FUNCTION_BLOCK DataTypesInteger (* Template for an empty basic function block *)
  (* Standard: 61499-2; Description: Normal just propagates the input to the output Max: sets to the highest possible value Min: sets to the lowest possible value Internal: sets the output from inside Copyright (c) 2019 Jan Holzweber This program and the accompanying materials are made available under the terms of the Eclipse Public License 2.0 which is available at https://www.eclipse.org/legal/epl-2.0/ SPDX-License-Identifier: EPL-2.0 *)
  (* Version 1.0, 2019-06-05, jholz *)
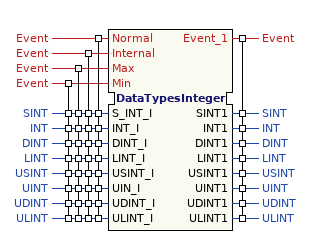
  EVENT_INPUT
    Normal WITH S_INT_I, INT_I, DINT_I, LINT_I, USINT_I, UIN_I, UDINT_I, ULINT_I;
    Internal WITH S_INT_I, INT_I, DINT_I, LINT_I, USINT_I, UIN_I, UDINT_I, ULINT_I;
    Max WITH S_INT_I, INT_I, DINT_I, LINT_I, USINT_I, UIN_I, UDINT_I, ULINT_I;
    Min WITH INT_I, S_INT_I, DINT_I, LINT_I, USINT_I, UIN_I, UDINT_I, ULINT_I;
  END_EVENT
  EVENT_OUTPUT
    Event_1 WITH SINT1, INT1, DINT1, LINT1, USINT1, UINT1, UDINT1, ULINT1;
  END_EVENT
  VAR_INPUT
    S_INT_I : SINT;
    INT_I : INT;
    DINT_I : DINT;
    LINT_I : LINT;
    USINT_I : USINT;
    UIN_I : UINT;
    UDINT_I : UDINT;
    ULINT_I : ULINT;
  END_VAR
  VAR_OUTPUT
    SINT1 : SINT;
    INT1 : INT;
    DINT1 : DINT;
    LINT1 : LINT;
    USINT1 : USINT;
    UINT1 : UINT;
    UDINT1 : UDINT;
    ULINT1 : ULINT;
  END_VAR
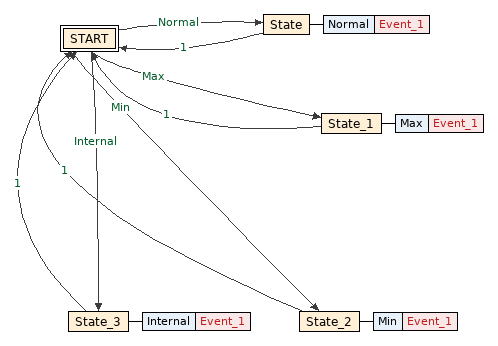
  EC_STATES
    START; (* Initial State *)
    State : Normal -> Event_1;
    State_1 : Max -> Event_1;
    State_2 : Min -> Event_1;
    State_3 : Internal -> Event_1;
  END_STATES
  EC_TRANSITIONS
    START TO State := Normal;
    State TO START := 1;
    START TO State_1 := Max;
    State_1 TO START := 1;
    START TO State_2 := Min;
    State_2 TO START := 1;
    START TO State_3 := Internal;
    State_3 TO START := 1;
  END_TRANSITIONS
  ALGORITHM Normal IN ST: (* new algorithm *)
SINT1 :=S_INT_I;
INT1:=INT_I;
DINT1:=DINT_I;
LINT1:=LINT_I;
USINT1:=USINT_I;
UINT1:=UIN_I;
UDINT1:=UDINT_I;
ULINT1:=ULINT_I;
  END_ALGORITHM
  ALGORITHM Max IN ST: (* new algorithm *)
SINT1 :=127;
INT1:=32767;
DINT1:=2147483647;
LINT1:=9223372036854775807;
USINT1:=255;
UINT1:=65535;
UDINT1:=4294967295;
ULINT1:=1;
  END_ALGORITHM
  ALGORITHM Min IN ST: (* new algorithm *)
SINT1 :=-128;
INT1:=-32768;
DINT1:=-2147483648;
LINT1:=-9223372036854775808;
USINT1:=0;
UINT1:=0;
UDINT1:=0;
ULINT1:=0;
  END_ALGORITHM
  ALGORITHM Internal IN ST: (* new algorithm *)
SINT1 :=-10;
INT1:=-20;
DINT1:=-30;
LINT1:=-40;
USINT1:=50;
UINT1:=60;
UDINT1:=70;
ULINT1:=80;
  END_ALGORITHM
END_FUNCTION_BLOCK
